FUNCTION_BLOCK EcMasterDeviceState IMPLEMENTS IEcTask
VAR_INPUT
END_VAR
VAR_OUTPUT
END_VAR
VAR
	iState : INT;
	masterDeviceState : Tc2_EtherCAT.FB_EcGetMasterDevState;
	_execute: BOOL;
	_done: BOOL;
	_busy: BOOL;
	_error: BOOL;
	_netId: AMSNETID;
END_VAR

CASE iState OF
	0:
		IF _execute THEN
			_done := FALSE;
			_busy := TRUE;
			_error := FALSE;
			masterDeviceState.bExecute := TRUE;
			IF masterDeviceState.bBusy THEN
				iState := 10;
				_execute := false;
			END_IF
		END_IF
	10:
		IF NOT masterDeviceState.bBusy THEN
			IF NOT masterDeviceState.bError THEN
				_done := TRUE;
			ELSE
				_error := TRUE;
			END_IF
			_busy := FALSE;
			masterDeviceState.bExecute := FALSE;
			iState := 0;
		END_IF
END_CASE

masterDeviceState(sNetId := Tc2_System.F_CreateAmsNetId(nIds := NetId));

{warning 'add method implementation '}
METHOD Abort : BOOL
masterDeviceState.bExecute := FALSE;
_busy := FALSE;
_execute := FALSE;
Abort := TRUE;
iState := 0;
END_METHOD

{warning 'add property implementation'}
PROPERTY Busy : BOOL
GET
Busy := _busy;
END_GET
END_PROPERTY

{warning 'add property implementation'}
PROPERTY Done : BOOL
GET
Done := _done;
END_GET
END_PROPERTY

{warning 'add property implementation'}
PROPERTY Error : BOOL
GET
Error := _error;
END_GET
END_PROPERTY

{warning 'add method implementation '}
METHOD Execute : BOOL
IF NOT masterDeviceState.bBusy THEN
	Execute := _execute := true;
END_IF
END_METHOD

PROPERTY MasterDevState : word
GET
MasterDevState := masterDeviceState.nDevState;
END_GET
END_PROPERTY

{warning 'add property implementation'}
PROPERTY NetID : amsnetid
GET
NetID := _netId;
END_GET
SET
_netId := NetID;
END_SET
END_PROPERTY

END_FUNCTION_BLOCK

(* stored: Version 1.1.0.1, ProductVersion 3.1.4024.11
   POU EcMasterDeviceState: Id {6c0f1c0f-9074-4eda-a761-d2f9a6c852a4}, SpecialFunc None
   Method Abort: Id {96926d07-0cbe-4cdf-ae17-a9cd6bae7911}
   Property Busy: Id {470b34dc-34eb-42b9-96fc-9e1cb423fd29}
   Get Get: Id {0c0b2877-09cf-4b16-9ecd-957b9fb1cb0f}
   Property Done: Id {e785ffb3-dfa6-4c3c-8771-fe02f2ac362b}
   Get Get: Id {59a52a93-c740-452d-a385-6367585644b6}
   Property Error: Id {25b38cea-6c0f-4e57-b6b0-43ff2aa7ac2f}
   Get Get: Id {859f7ed7-6946-41c2-999f-5a32c7ec37b7}
   Method Execute: Id {04c3b097-9e4a-450b-9090-c61b4c87f835}
   Property MasterDevState: Id {6236fa1e-698c-44ce-86f5-59487ba54c23}
   Get Get: Id {0ac15539-9de6-46a2-97fc-2a473650aada}
   Property NetID: Id {55123738-a8aa-48a5-9828-bb983bf71021}
   Get Get: Id {0338a1d1-aade-4a5d-959e-701e10bfa219}
   Set Set: Id {181b8b0e-df13-4014-87d4-994487d06e71} *)
